(* Logix 5000 project; controller cal1615 1756-L62 rev 20.19; software revision 20.05; part 39 of 81 *)
(* tags used below, declared in another part *)
   FAULT : BOOL;   // Fault AFI
   HMI : BOOL;   // AFI HMI
   p01_ai_lc_4 : REAL;
   p01r09_pb_global_reset : BOOL;   // System Modes PB: Global Fault Reset
   p02_real_from_hmi : hmi_real;   // MOP HMI Iface Real from HMI
   p20_acc_fill_time_sec : REAL;   // Letoff Accumulator Fill Time
   p20_ai_lc01 : REAL;   // Letoff Analog Input Line Tension Load Cell Splicer
   p20_ai_letoff_dia : REAL;   // Letoff Analog Inputs Letoff Roll Diameter [in]
   p20_ai_lo_turret_amps : REAL;   // Letoff Inputs Letoff Turret VFD Amps
   p20_ai_lo_turret_hz : REAL;   // Letoff Inputs Letoff Turret VFD Hz
   p20_ai_lo_turret_speed : REAL;
   p20_ai_loa_speed : REAL;   // Letoff Inputs Letoff A VFD Surface Speed
   p20_ai_lob_speed : REAL;   // Letoff Inputs Letoff A Speed
   p20_ao_acc_ctr_prs : REAL;   // Letoff Analog Output Accumulator Counter Pressure
   p20_ao_acc_fill_prs : REAL;   // Letoff Analog Output Accumulator Fill Pressure
   p20_ao_acc_ten_prs : REAL;   // Letoff Analog Output Accumulator Tension Pressure
   p20_ao_loa_selected_speed : REAL;   // Letoff Output Selected Speed
   p20_di_clutch_prs_ok : BOOL;   // Letoff Modes Accumulator Position Mode
   p20_dint_to_hmi : DINT[16];   // Letoff Dint to HMI
   p20_loa_ai_amps : REAL;   // Letoff Inputs Letoff A VFD Amps
   p20_loa_ai_hz : REAL;   // Letoff Inputs Letoff A Hz
   p20_lob_ai_amps : REAL;   // Letoff Inputs Letoff B VFD Amps
   p20_lob_ai_hz : REAL;   // Letoff Inputs Letoff B VFD Hz
   p20_real_to_hmi : REAL[112];   // Letoff Real to HMI
   p20r01 : routine;   // Letoff Main
   p20r06 : routine;   // Letoff Real to HMI
   p20r06_ave_lc : REAL;
   p20r06_lc_ave_ctrl : CONTROL;
   p20r06_lc_buffer : REAL[20];
   p20r06_lc_ctrl : CONTROL;
   p20r06_sample_timer : TIMER;
   p20r06_timer_fault : TIMER[4];   // Letoff Real to HMI Fault Delay
   p20r06_timer_warning : TIMER[4];   // Letoff Real to HMI Warning Delay
   p20r06_unload : DINT;
   p20r07 : routine;   // Letoff Alarms
   p20r07_timer_fault : TIMER[4];   // Letoff Alarms Fault Delay
   p20r07_timer_warning : TIMER[4];   // Letoff Alarms Warning Delay
   p20r08 : routine;   // Letoff Warnings
   p20r08_timer_fault : TIMER[4];   // Letoff Warnings Fault Delay
   p20r08_timer_warning : TIMER[4];   // Letoff Warnings Warning Delay
   p20r10_pid_tens_cv : REAL;   // Letoff Letoff Speed Control Control Value CV
   p20r13_ai_acc_pct : REAL;   // Letoff Accumulator Pct Full
   p20r13_ai_loa_footage_ft : REAL;
   p20r13_ai_lob_footage_ft : REAL;
   p20r15 : routine;   // Letoff Letoff A VFD
   p20r16 : routine;   // Letoff Letoff B VFD
   p20r18 : routine;   // Letoff Letoff Turret VFD
(* P20_Letoff, continued *)

ROUTINE R06_Real_to_HMI   (* ladder *)
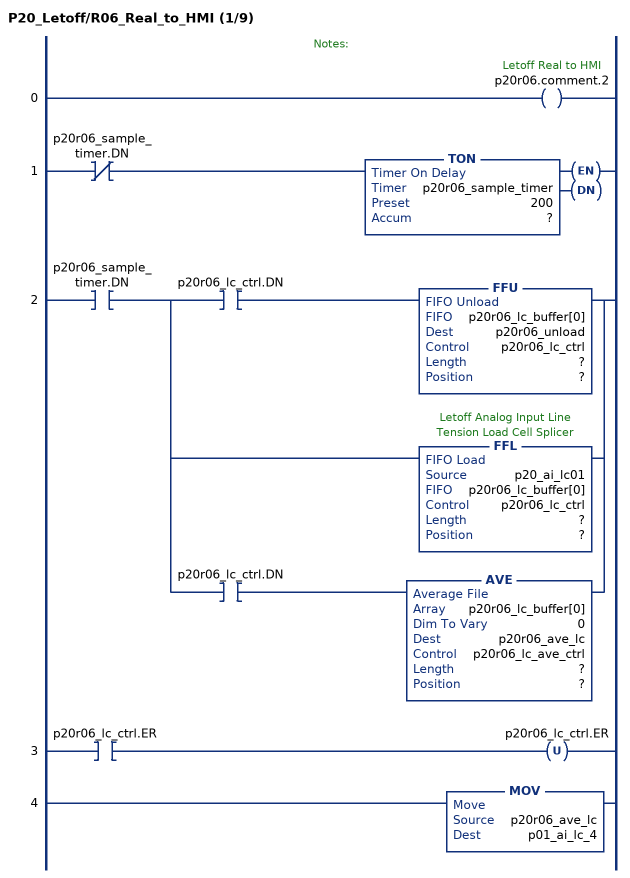
   // Notes:
   0: OTE(p20r06.comment.2);
   1: XIO(p20r06_sample_timer.DN)TON(p20r06_sample_timer,?,?);
   2: XIC(p20r06_sample_timer.DN)[XIC(p20r06_lc_ctrl.DN) FFU(p20r06_lc_buffer[0],p20r06_unload,p20r06_lc_ctrl,?,?) ,FFL(p20_ai_lc01,p20r06_lc_buffer[0],p20r06_lc_ctrl,?,?) ,XIC(p20r06_lc_ctrl.DN) AVE(p20r06_lc_buffer[0],0,p20r06_ave_lc,p20r06_lc_ave_ctrl,?,?) ];
   3: XIC(p20r06_lc_ctrl.ER)OTU(p20r06_lc_ctrl.ER);
   4: MOV(p20r06_ave_lc,p01_ai_lc_4);
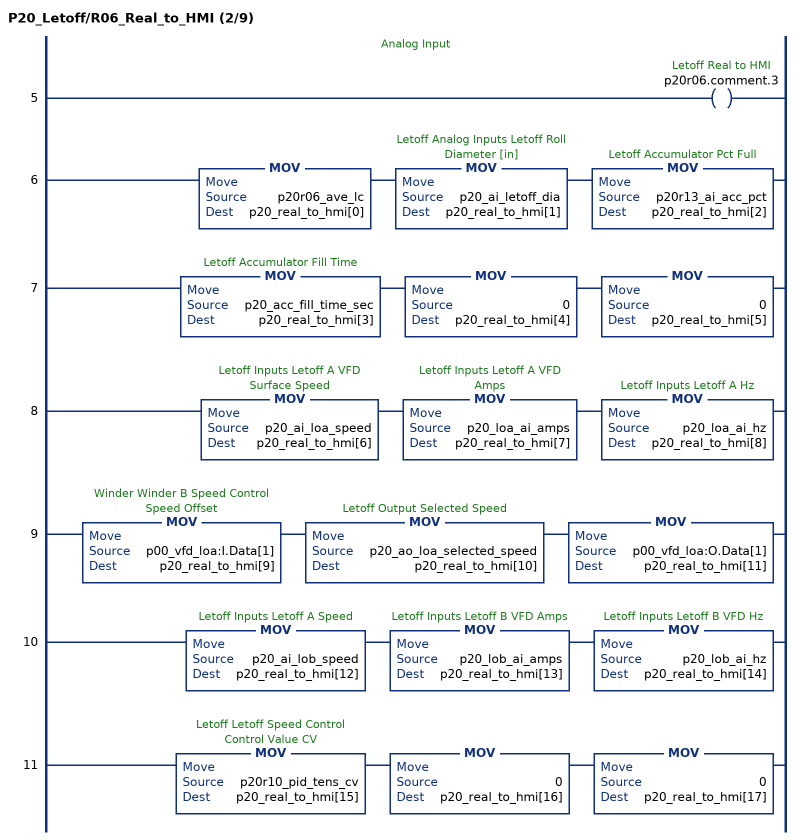
   // Analog Input
   5: OTE(p20r06.comment.3);
   6: MOV(p20r06_ave_lc,p20_real_to_hmi[0])MOV(p20_ai_letoff_dia,p20_real_to_hmi[1])MOV(p20r13_ai_acc_pct,p20_real_to_hmi[2]);
   7: MOV(p20_acc_fill_time_sec,p20_real_to_hmi[3])MOV(0,p20_real_to_hmi[4])MOV(0,p20_real_to_hmi[5]);
   8: MOV(p20_ai_loa_speed,p20_real_to_hmi[6])MOV(p20_loa_ai_amps,p20_real_to_hmi[7])MOV(p20_loa_ai_hz,p20_real_to_hmi[8]);
   9: MOV(p00_vfd_loa:I.Data[1],p20_real_to_hmi[9])MOV(p20_ao_loa_selected_speed,p20_real_to_hmi[10])MOV(p00_vfd_loa:O.Data[1],p20_real_to_hmi[11]);
   10: MOV(p20_ai_lob_speed,p20_real_to_hmi[12])MOV(p20_lob_ai_amps,p20_real_to_hmi[13])MOV(p20_lob_ai_hz,p20_real_to_hmi[14]);
   11: MOV(p20r10_pid_tens_cv,p20_real_to_hmi[15])MOV(0,p20_real_to_hmi[16])MOV(0,p20_real_to_hmi[17]);
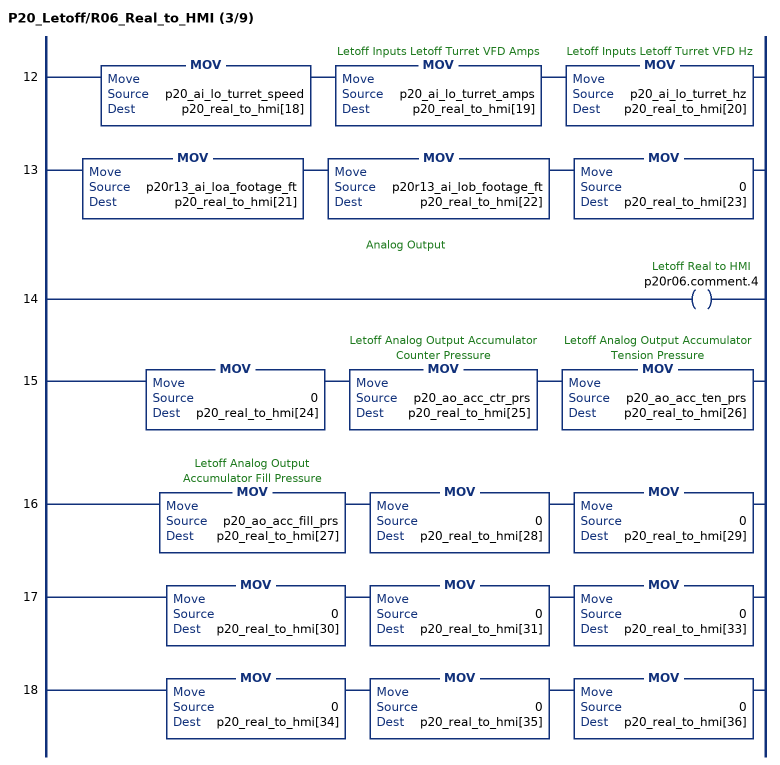
   12: MOV(p20_ai_lo_turret_speed,p20_real_to_hmi[18])MOV(p20_ai_lo_turret_amps,p20_real_to_hmi[19])MOV(p20_ai_lo_turret_hz,p20_real_to_hmi[20]);
   13: MOV(p20r13_ai_loa_footage_ft,p20_real_to_hmi[21])MOV(p20r13_ai_lob_footage_ft,p20_real_to_hmi[22])MOV(0,p20_real_to_hmi[23]);
   // Analog Output
   14: OTE(p20r06.comment.4);
   15: MOV(0,p20_real_to_hmi[24])MOV(p20_ao_acc_ctr_prs,p20_real_to_hmi[25])MOV(p20_ao_acc_ten_prs,p20_real_to_hmi[26]);
   16: MOV(p20_ao_acc_fill_prs,p20_real_to_hmi[27])MOV(0,p20_real_to_hmi[28])MOV(0,p20_real_to_hmi[29]);
   17: MOV(0,p20_real_to_hmi[30])MOV(0,p20_real_to_hmi[31])MOV(0,p20_real_to_hmi[33]);
   18: MOV(0,p20_real_to_hmi[34])MOV(0,p20_real_to_hmi[35])MOV(0,p20_real_to_hmi[36]);
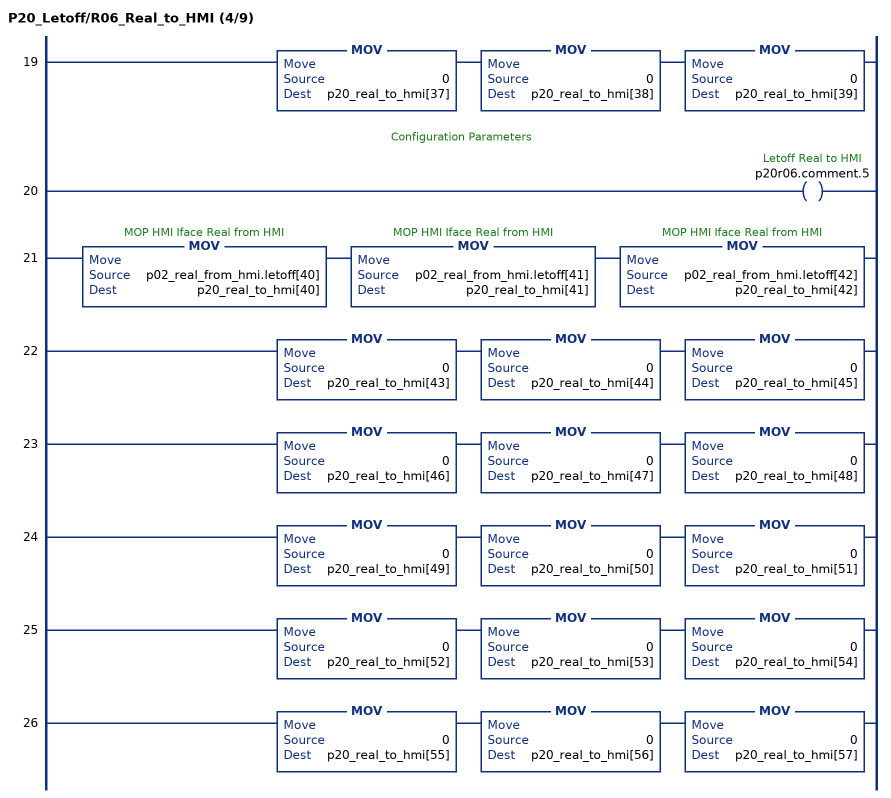
   19: MOV(0,p20_real_to_hmi[37])MOV(0,p20_real_to_hmi[38])MOV(0,p20_real_to_hmi[39]);
   // Configuration Parameters
   20: OTE(p20r06.comment.5);
   21: MOV(p02_real_from_hmi.letoff[40],p20_real_to_hmi[40])MOV(p02_real_from_hmi.letoff[41],p20_real_to_hmi[41])MOV(p02_real_from_hmi.letoff[42],p20_real_to_hmi[42]);
   22: MOV(0,p20_real_to_hmi[43])MOV(0,p20_real_to_hmi[44])MOV(0,p20_real_to_hmi[45]);
   23: MOV(0,p20_real_to_hmi[46])MOV(0,p20_real_to_hmi[47])MOV(0,p20_real_to_hmi[48]);
   24: MOV(0,p20_real_to_hmi[49])MOV(0,p20_real_to_hmi[50])MOV(0,p20_real_to_hmi[51]);
   25: MOV(0,p20_real_to_hmi[52])MOV(0,p20_real_to_hmi[53])MOV(0,p20_real_to_hmi[54]);
   26: MOV(0,p20_real_to_hmi[55])MOV(0,p20_real_to_hmi[56])MOV(0,p20_real_to_hmi[57]);
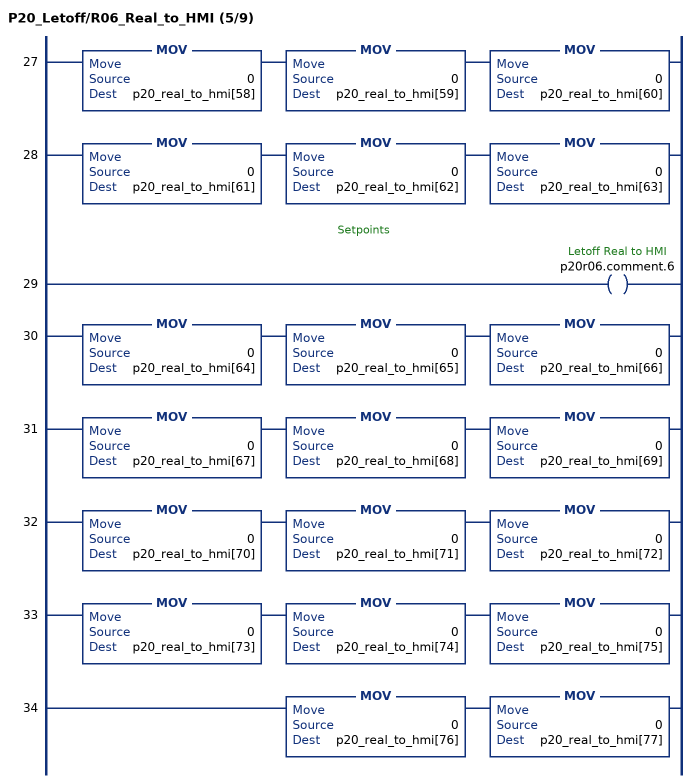
   27: MOV(0,p20_real_to_hmi[58])MOV(0,p20_real_to_hmi[59])MOV(0,p20_real_to_hmi[60]);
   28: MOV(0,p20_real_to_hmi[61])MOV(0,p20_real_to_hmi[62])MOV(0,p20_real_to_hmi[63]);
   // Setpoints
   29: OTE(p20r06.comment.6);
   30: MOV(0,p20_real_to_hmi[64])MOV(0,p20_real_to_hmi[65])MOV(0,p20_real_to_hmi[66]);
   31: MOV(0,p20_real_to_hmi[67])MOV(0,p20_real_to_hmi[68])MOV(0,p20_real_to_hmi[69]);
   32: MOV(0,p20_real_to_hmi[70])MOV(0,p20_real_to_hmi[71])MOV(0,p20_real_to_hmi[72]);
   33: MOV(0,p20_real_to_hmi[73])MOV(0,p20_real_to_hmi[74])MOV(0,p20_real_to_hmi[75]);
   34: MOV(0,p20_real_to_hmi[76])MOV(0,p20_real_to_hmi[77]);
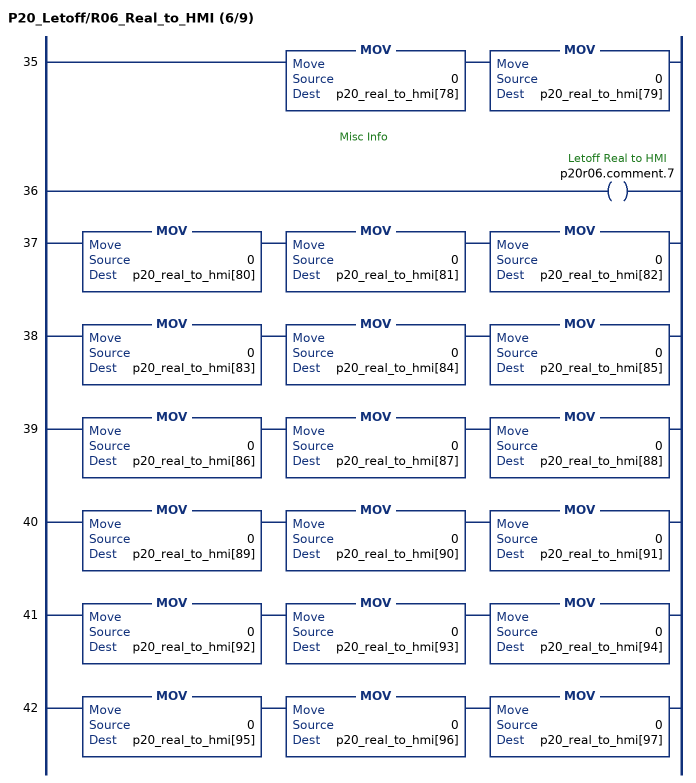
   35: MOV(0,p20_real_to_hmi[78])MOV(0,p20_real_to_hmi[79]);
   // Misc Info
   36: OTE(p20r06.comment.7);
   37: MOV(0,p20_real_to_hmi[80])MOV(0,p20_real_to_hmi[81])MOV(0,p20_real_to_hmi[82]);
   38: MOV(0,p20_real_to_hmi[83])MOV(0,p20_real_to_hmi[84])MOV(0,p20_real_to_hmi[85]);
   39: MOV(0,p20_real_to_hmi[86])MOV(0,p20_real_to_hmi[87])MOV(0,p20_real_to_hmi[88]);
   40: MOV(0,p20_real_to_hmi[89])MOV(0,p20_real_to_hmi[90])MOV(0,p20_real_to_hmi[91]);
   41: MOV(0,p20_real_to_hmi[92])MOV(0,p20_real_to_hmi[93])MOV(0,p20_real_to_hmi[94]);
   42: MOV(0,p20_real_to_hmi[95])MOV(0,p20_real_to_hmi[96])MOV(0,p20_real_to_hmi[97]);
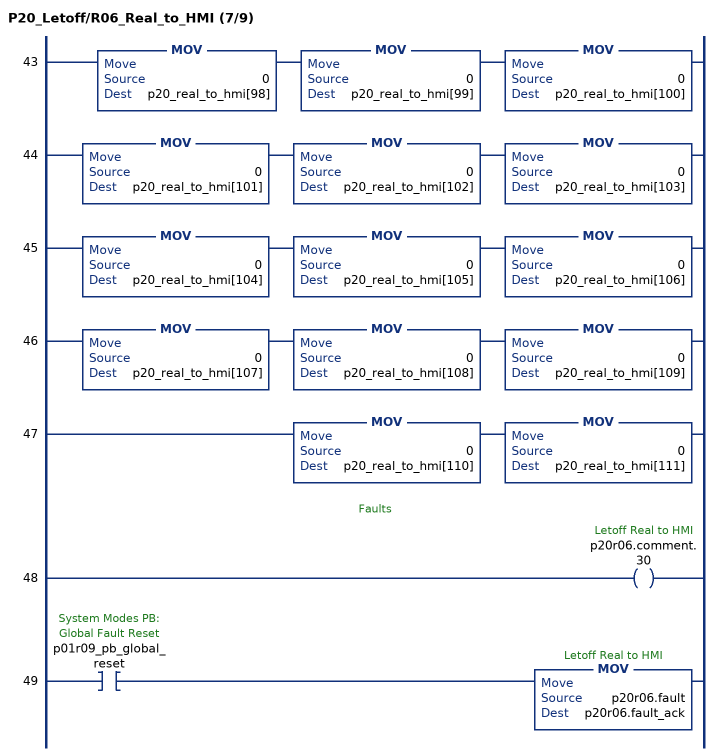
   43: MOV(0,p20_real_to_hmi[98])MOV(0,p20_real_to_hmi[99])MOV(0,p20_real_to_hmi[100]);
   44: MOV(0,p20_real_to_hmi[101])MOV(0,p20_real_to_hmi[102])MOV(0,p20_real_to_hmi[103]);
   45: MOV(0,p20_real_to_hmi[104])MOV(0,p20_real_to_hmi[105])MOV(0,p20_real_to_hmi[106]);
   46: MOV(0,p20_real_to_hmi[107])MOV(0,p20_real_to_hmi[108])MOV(0,p20_real_to_hmi[109]);
   47: MOV(0,p20_real_to_hmi[110])MOV(0,p20_real_to_hmi[111]);
   // Faults
   48: OTE(p20r06.comment.30);
   49: XIC(p01r09_pb_global_reset)MOV(p20r06.fault,p20r06.fault_ack);
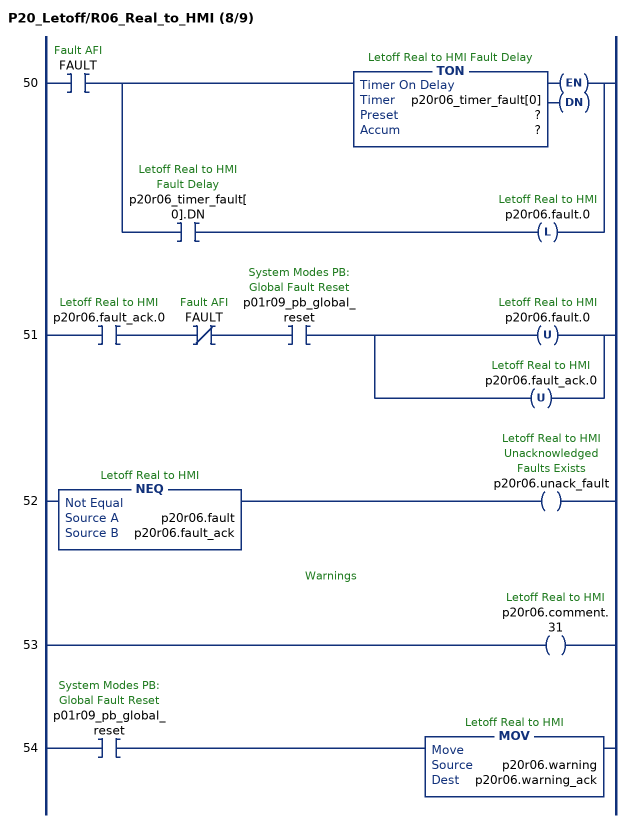
   50: XIC(FAULT)[TON(p20r06_timer_fault[0],?,?) ,XIC(p20r06_timer_fault[0].DN) OTL(p20r06.fault.0) ];
   51: XIC(p20r06.fault_ack.0)XIO(FAULT)XIC(p01r09_pb_global_reset)[OTU(p20r06.fault.0) ,OTU(p20r06.fault_ack.0) ];
   52: NEQ(p20r06.fault,p20r06.fault_ack)OTE(p20r06.unack_fault);
   // Warnings
   53: OTE(p20r06.comment.31);
   54: XIC(p01r09_pb_global_reset)MOV(p20r06.warning,p20r06.warning_ack);
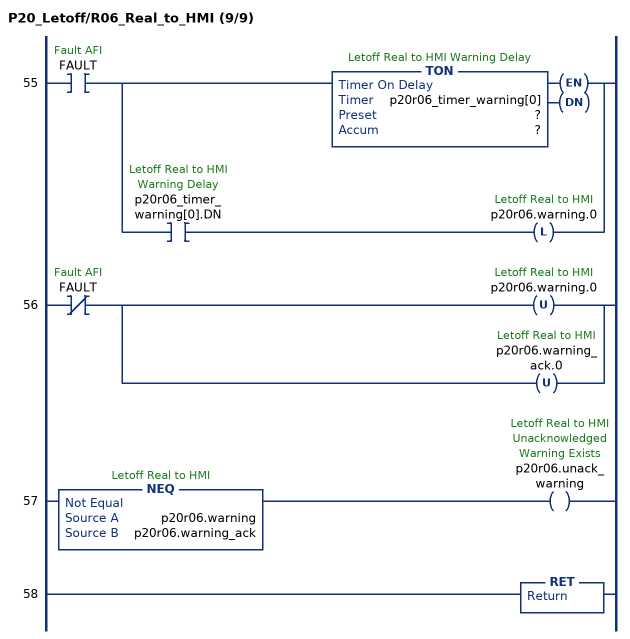
   55: XIC(FAULT)[TON(p20r06_timer_warning[0],?,?) ,XIC(p20r06_timer_warning[0].DN) OTL(p20r06.warning.0) ];
   56: XIO(FAULT)[OTU(p20r06.warning.0) ,OTU(p20r06.warning_ack.0) ];
   57: NEQ(p20r06.warning,p20r06.warning_ack)OTE(p20r06.unack_warning);
   58: RET();
END_ROUTINE

ROUTINE R07_Alarms   (* ladder *)
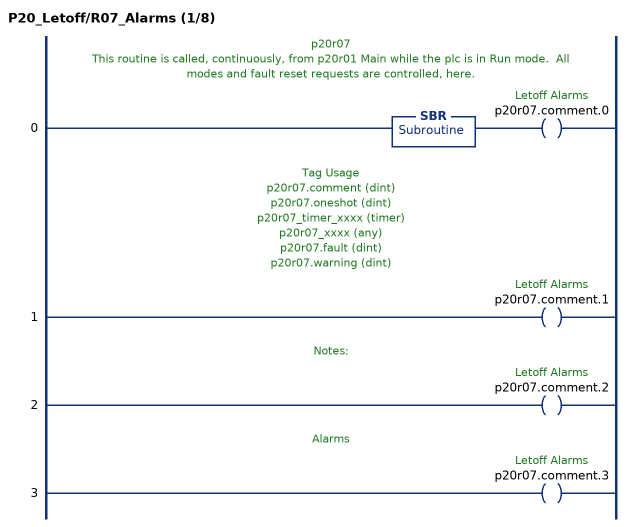
   // p20r07
   // This routine is called, continuously, from p20r01 Main while the plc is in Run mode.  All modes and fault reset requests are controlled, here.
   0: SBR()OTE(p20r07.comment.0);
   // Tag Usage
   // p20r07.comment (dint)
   // p20r07.oneshot (dint)
   // p20r07_timer_xxxx (timer)
   // p20r07_xxxx (any)
   // p20r07.fault (dint)
   // p20r07.warning (dint)
   1: OTE(p20r07.comment.1);
   // Notes:
   2: OTE(p20r07.comment.2);
   // Alarms
   3: OTE(p20r07.comment.3);
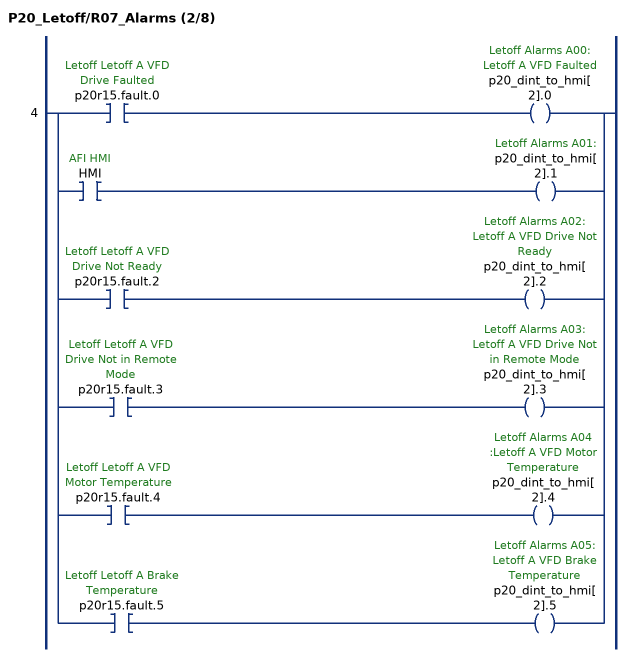
   4: [XIC(p20r15.fault.0) OTE(p20_dint_to_hmi[2].0) ,XIC(HMI) OTE(p20_dint_to_hmi[2].1) ,XIC(p20r15.fault.2) OTE(p20_dint_to_hmi[2].2) ,XIC(p20r15.fault.3) OTE(p20_dint_to_hmi[2].3) ,XIC(p20r15.fault.4) OTE(p20_dint_to_hmi[2].4) ,XIC(p20r15.fault.5) OTE(p20_dint_to_hmi[2].5) ];
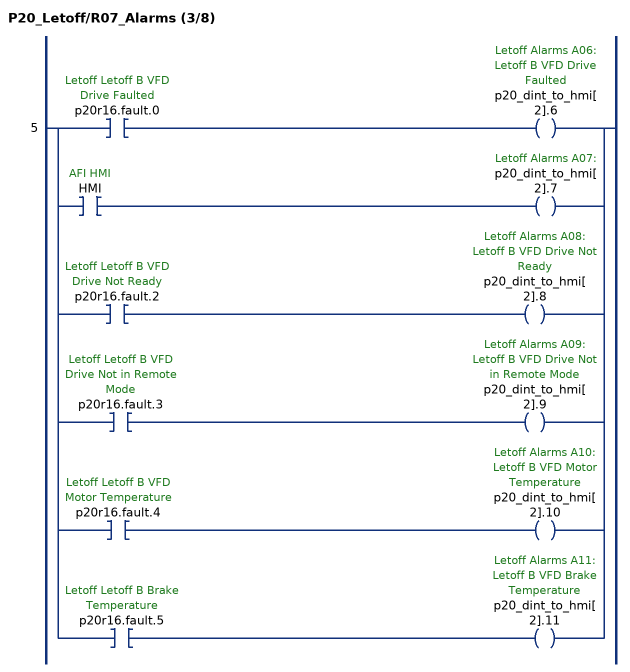
   5: [XIC(p20r16.fault.0) OTE(p20_dint_to_hmi[2].6) ,XIC(HMI) OTE(p20_dint_to_hmi[2].7) ,XIC(p20r16.fault.2) OTE(p20_dint_to_hmi[2].8) ,XIC(p20r16.fault.3) OTE(p20_dint_to_hmi[2].9) ,XIC(p20r16.fault.4) OTE(p20_dint_to_hmi[2].10) ,XIC(p20r16.fault.5) OTE(p20_dint_to_hmi[2].11) ];
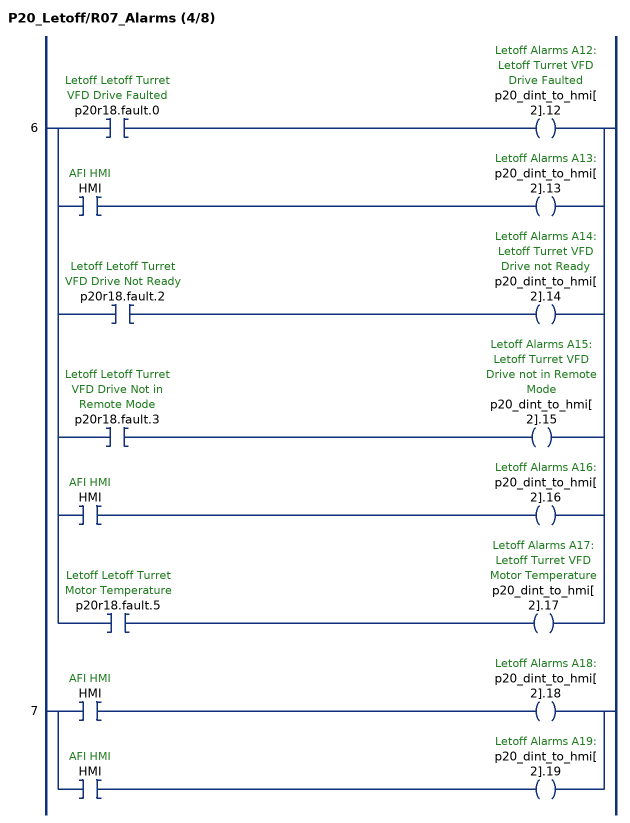
   6: [XIC(p20r18.fault.0) OTE(p20_dint_to_hmi[2].12) ,XIC(HMI) OTE(p20_dint_to_hmi[2].13) ,XIC(p20r18.fault.2) OTE(p20_dint_to_hmi[2].14) ,XIC(p20r18.fault.3) OTE(p20_dint_to_hmi[2].15) ,XIC(HMI) OTE(p20_dint_to_hmi[2].16) ,XIC(p20r18.fault.5) OTE(p20_dint_to_hmi[2].17) ];
   7: [XIC(HMI) OTE(p20_dint_to_hmi[2].18) ,XIC(HMI) OTE(p20_dint_to_hmi[2].19) ];
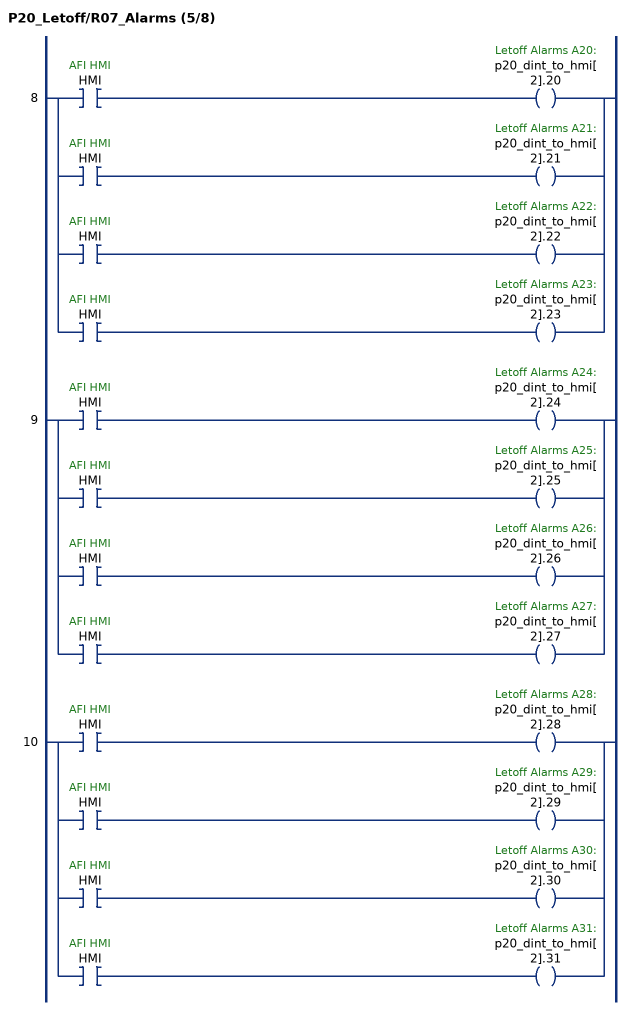
   8: [XIC(HMI) OTE(p20_dint_to_hmi[2].20) ,XIC(HMI) OTE(p20_dint_to_hmi[2].21) ,XIC(HMI) OTE(p20_dint_to_hmi[2].22) ,XIC(HMI) OTE(p20_dint_to_hmi[2].23) ];
   9: [XIC(HMI) OTE(p20_dint_to_hmi[2].24) ,XIC(HMI) OTE(p20_dint_to_hmi[2].25) ,XIC(HMI) OTE(p20_dint_to_hmi[2].26) ,XIC(HMI) OTE(p20_dint_to_hmi[2].27) ];
   10: [XIC(HMI) OTE(p20_dint_to_hmi[2].28) ,XIC(HMI) OTE(p20_dint_to_hmi[2].29) ,XIC(HMI) OTE(p20_dint_to_hmi[2].30) ,XIC(HMI) OTE(p20_dint_to_hmi[2].31) ];
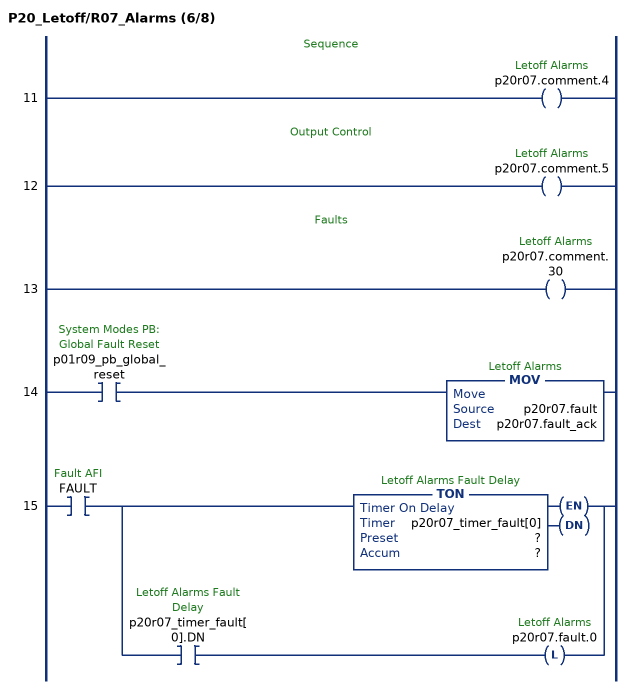
   // Sequence
   11: OTE(p20r07.comment.4);
   // Output Control
   12: OTE(p20r07.comment.5);
   // Faults
   13: OTE(p20r07.comment.30);
   14: XIC(p01r09_pb_global_reset)MOV(p20r07.fault,p20r07.fault_ack);
   15: XIC(FAULT)[TON(p20r07_timer_fault[0],?,?) ,XIC(p20r07_timer_fault[0].DN) OTL(p20r07.fault.0) ];
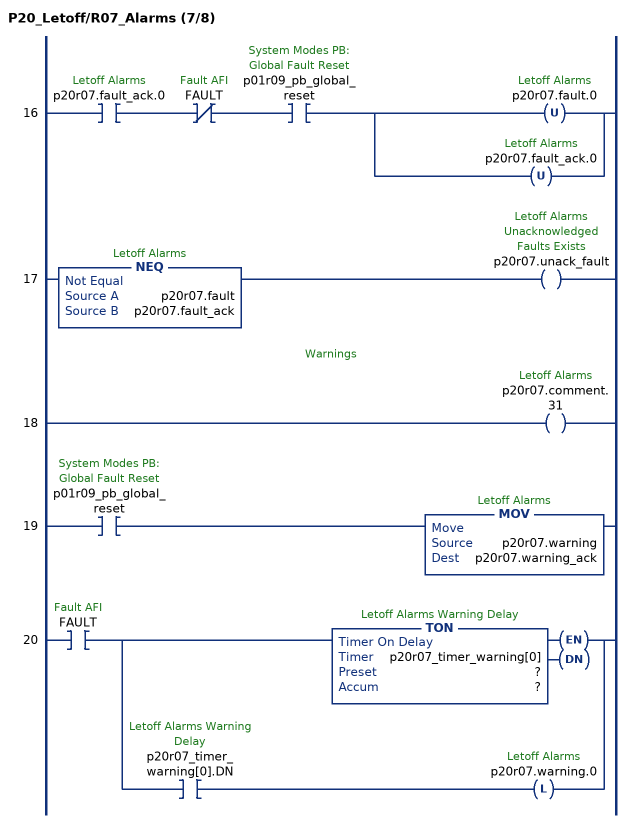
   16: XIC(p20r07.fault_ack.0)XIO(FAULT)XIC(p01r09_pb_global_reset)[OTU(p20r07.fault.0) ,OTU(p20r07.fault_ack.0) ];
   17: NEQ(p20r07.fault,p20r07.fault_ack)OTE(p20r07.unack_fault);
   // Warnings
   18: OTE(p20r07.comment.31);
   19: XIC(p01r09_pb_global_reset)MOV(p20r07.warning,p20r07.warning_ack);
   20: XIC(FAULT)[TON(p20r07_timer_warning[0],?,?) ,XIC(p20r07_timer_warning[0].DN) OTL(p20r07.warning.0) ];
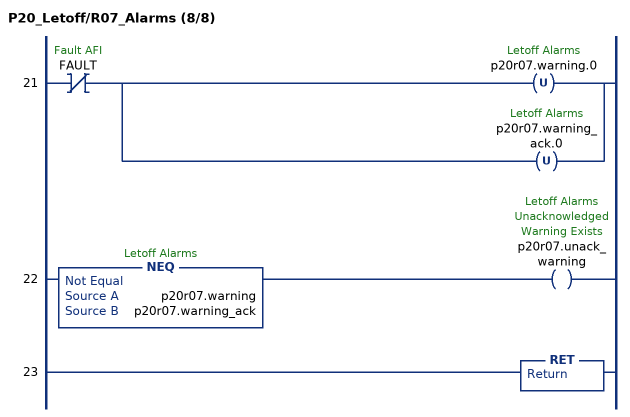
   21: XIO(FAULT)[OTU(p20r07.warning.0) ,OTU(p20r07.warning_ack.0) ];
   22: NEQ(p20r07.warning,p20r07.warning_ack)OTE(p20r07.unack_warning);
   23: RET();
END_ROUTINE

ROUTINE R08_Warnings   (* ladder *)
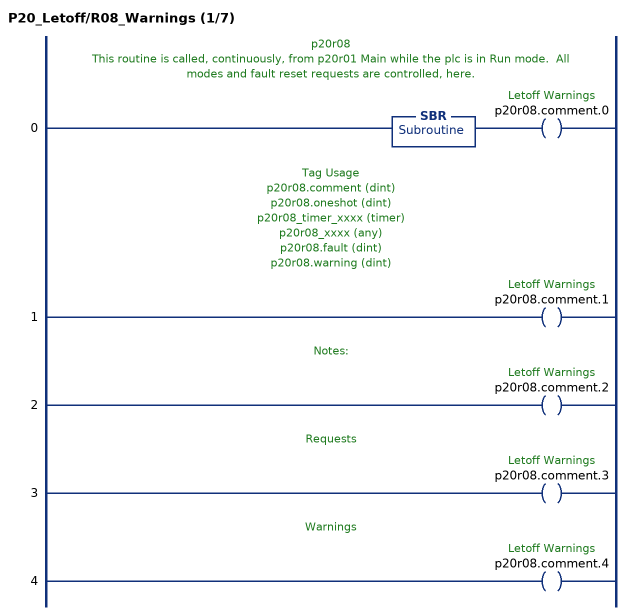
   // p20r08
   // This routine is called, continuously, from p20r01 Main while the plc is in Run mode.  All modes and fault reset requests are controlled, here.
   0: SBR()OTE(p20r08.comment.0);
   // Tag Usage
   // p20r08.comment (dint)
   // p20r08.oneshot (dint)
   // p20r08_timer_xxxx (timer)
   // p20r08_xxxx (any)
   // p20r08.fault (dint)
   // p20r08.warning (dint)
   1: OTE(p20r08.comment.1);
   // Notes:
   2: OTE(p20r08.comment.2);
   // Requests
   3: OTE(p20r08.comment.3);
   // Warnings
   4: OTE(p20r08.comment.4);
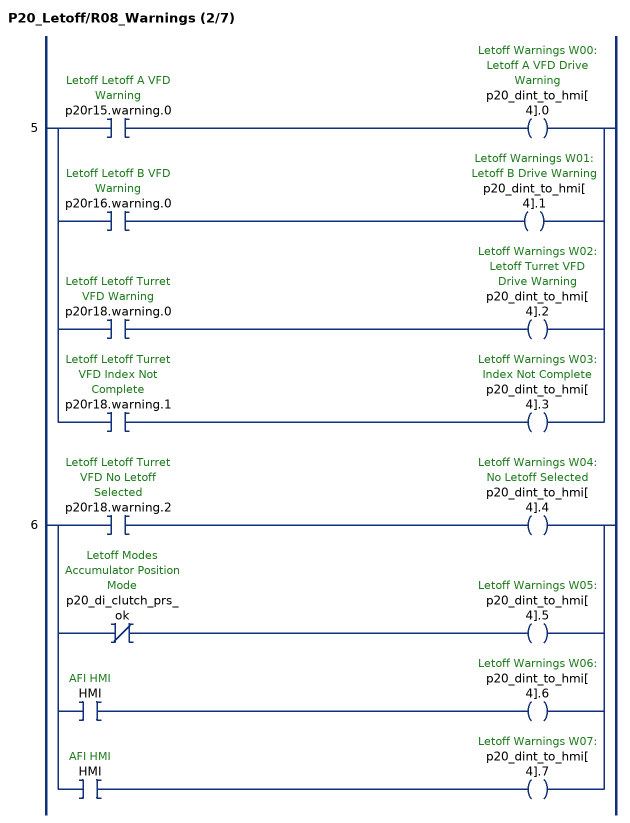
   5: [XIC(p20r15.warning.0) OTE(p20_dint_to_hmi[4].0) ,XIC(p20r16.warning.0) OTE(p20_dint_to_hmi[4].1) ,XIC(p20r18.warning.0) OTE(p20_dint_to_hmi[4].2) ,XIC(p20r18.warning.1) OTE(p20_dint_to_hmi[4].3) ];
   6: [XIC(p20r18.warning.2) OTE(p20_dint_to_hmi[4].4) ,XIO(p20_di_clutch_prs_ok) OTE(p20_dint_to_hmi[4].5) ,XIC(HMI) OTE(p20_dint_to_hmi[4].6) ,XIC(HMI) OTE(p20_dint_to_hmi[4].7) ];
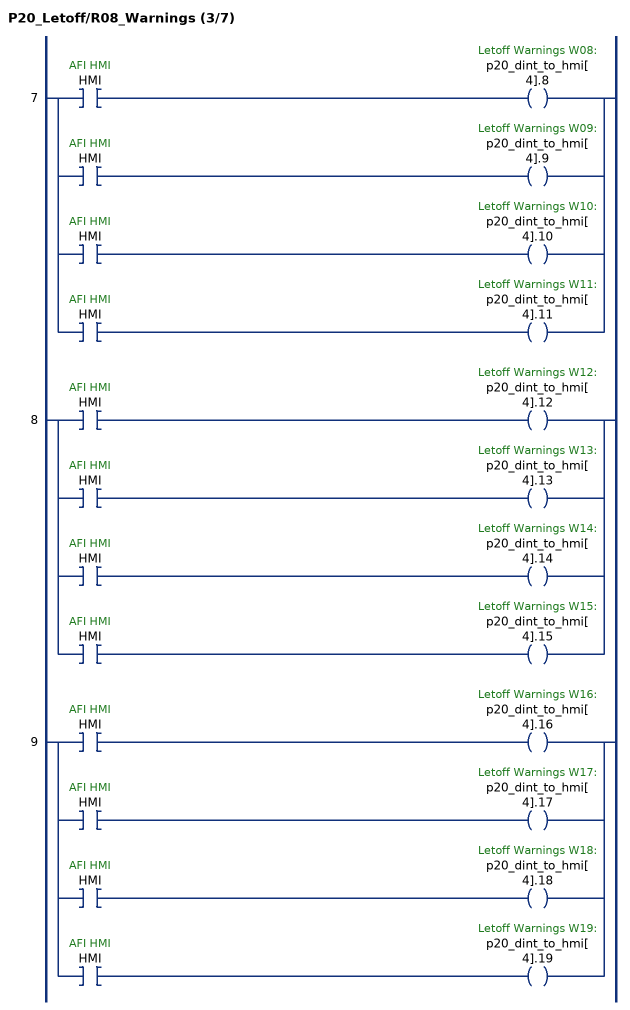
   7: [XIC(HMI) OTE(p20_dint_to_hmi[4].8) ,XIC(HMI) OTE(p20_dint_to_hmi[4].9) ,XIC(HMI) OTE(p20_dint_to_hmi[4].10) ,XIC(HMI) OTE(p20_dint_to_hmi[4].11) ];
   8: [XIC(HMI) OTE(p20_dint_to_hmi[4].12) ,XIC(HMI) OTE(p20_dint_to_hmi[4].13) ,XIC(HMI) OTE(p20_dint_to_hmi[4].14) ,XIC(HMI) OTE(p20_dint_to_hmi[4].15) ];
   9: [XIC(HMI) OTE(p20_dint_to_hmi[4].16) ,XIC(HMI) OTE(p20_dint_to_hmi[4].17) ,XIC(HMI) OTE(p20_dint_to_hmi[4].18) ,XIC(HMI) OTE(p20_dint_to_hmi[4].19) ];
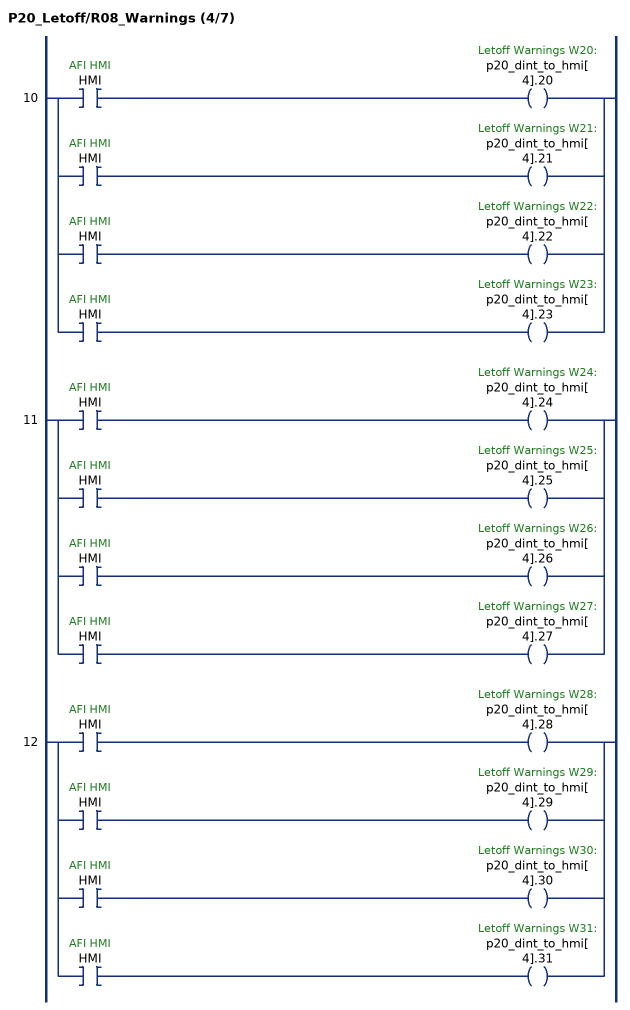
   10: [XIC(HMI) OTE(p20_dint_to_hmi[4].20) ,XIC(HMI) OTE(p20_dint_to_hmi[4].21) ,XIC(HMI) OTE(p20_dint_to_hmi[4].22) ,XIC(HMI) OTE(p20_dint_to_hmi[4].23) ];
   11: [XIC(HMI) OTE(p20_dint_to_hmi[4].24) ,XIC(HMI) OTE(p20_dint_to_hmi[4].25) ,XIC(HMI) OTE(p20_dint_to_hmi[4].26) ,XIC(HMI) OTE(p20_dint_to_hmi[4].27) ];
   12: [XIC(HMI) OTE(p20_dint_to_hmi[4].28) ,XIC(HMI) OTE(p20_dint_to_hmi[4].29) ,XIC(HMI) OTE(p20_dint_to_hmi[4].30) ,XIC(HMI) OTE(p20_dint_to_hmi[4].31) ];
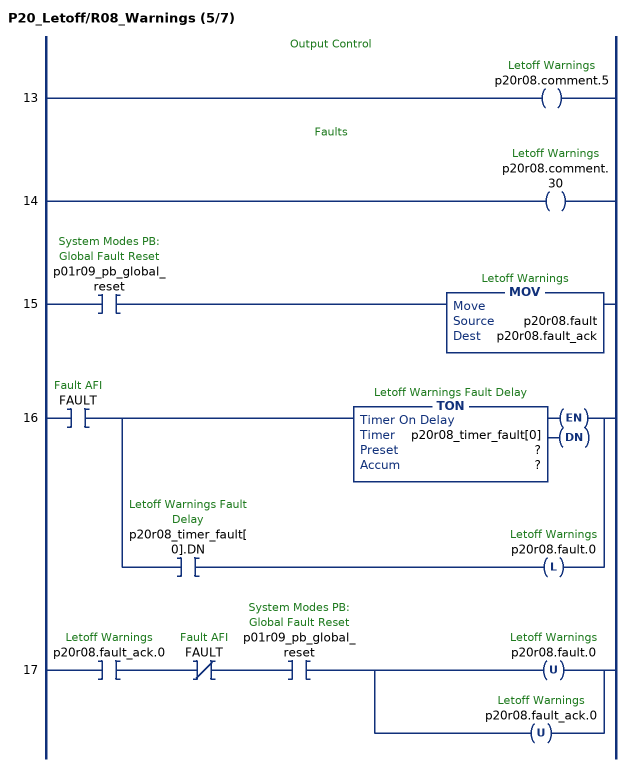
   // Output Control
   13: OTE(p20r08.comment.5);
   // Faults
   14: OTE(p20r08.comment.30);
   15: XIC(p01r09_pb_global_reset)MOV(p20r08.fault,p20r08.fault_ack);
   16: XIC(FAULT)[TON(p20r08_timer_fault[0],?,?) ,XIC(p20r08_timer_fault[0].DN) OTL(p20r08.fault.0) ];
   17: XIC(p20r08.fault_ack.0)XIO(FAULT)XIC(p01r09_pb_global_reset)[OTU(p20r08.fault.0) ,OTU(p20r08.fault_ack.0) ];
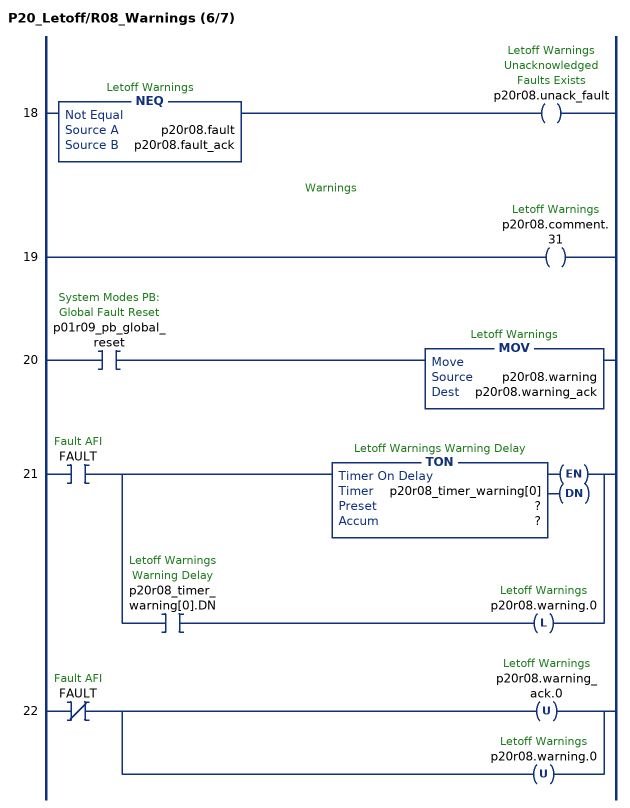
   18: NEQ(p20r08.fault,p20r08.fault_ack)OTE(p20r08.unack_fault);
   // Warnings
   19: OTE(p20r08.comment.31);
   20: XIC(p01r09_pb_global_reset)MOV(p20r08.warning,p20r08.warning_ack);
   21: XIC(FAULT)[TON(p20r08_timer_warning[0],?,?) ,XIC(p20r08_timer_warning[0].DN) OTL(p20r08.warning.0) ];
   22: XIO(FAULT)[OTU(p20r08.warning_ack.0) ,OTU(p20r08.warning.0) ];
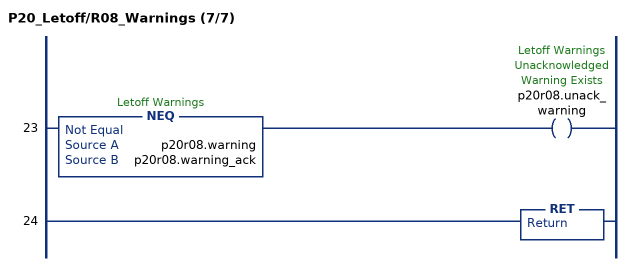
   23: NEQ(p20r08.warning,p20r08.warning_ack)OTE(p20r08.unack_warning);
   24: RET();
END_ROUTINE
